PROGRAM POU_SA01_ReadScanners
VAR
	
	LeftOuter				: BOOL;
	LeftInner				: BOOL; // Based on logic, could omit using inner scanners.
	RightOuter				: BOOL; // Based on logic, could omit using inner scanners.
	RightInner				: BOOL;
	
END_VAR

LeftOuter					:= R100_01;
LeftInner					:= R100_02; 
RightInner					:= R100_03; 
RightOuter					:= R100_04;

IF LeftOuter = TRUE THEN
	
	LeftLimitExceeded 		:= TRUE;
	
ELSE
	
	LeftLimitExceeded 		:= FALSE;
	
END_IF

IF RightOuter = TRUE THEN
	
	RightLimitExceeded 		:= TRUE;
	
ELSE
	
	RightLimitExceeded 		:= FALSE;
	
END_IF

END_PROGRAM

(* stored: Version 1.1.0.1, ProductVersion 3.1.4022.7
   POU POU_SA01_ReadScanners: Id {a1d13425-713e-4ee5-9a6a-45a4c7136efd}, SpecialFunc None *)
